# EPICS substitutions: apps/mpodLvApp/Db/mvtlv.substitutions
file "db/mpod8008l.db" {
    pattern {HOST,CH,SCAN,PORT,DETALIAS}
{"%(mvtlv)","0","2 second","B_HW_MVTLV_Sl0_Ch0","B_DET_MVT_LV_0"}
{"%(mvtlv)","1","2 second","B_HW_MVTLV_Sl0_Ch1","B_DET_MVT_LV_1"}
{"%(mvtlv)","2","2 second","B_HW_MVTLV_Sl0_Ch2","B_DET_MVT_LV_2"}
{"%(mvtlv)","3","2 second","B_HW_MVTLV_Sl0_Ch3","B_DET_MVT_LV_3"}
{"%(mvtlv)","4","2 second","B_HW_MVTLV_Sl0_Ch4","B_DET_MVT_LV_4"}
{"%(mvtlv)","5","2 second","B_HW_MVTLV_Sl0_Ch5","B_DET_MVT_LV_5"}
}
